TYPE ST_DivertConfig :
STRUCT
 	SwitchOpMode         						: E_SwitchOpMode;
	IntervalToDivert							: UDINT := 1;
	MaxAllowedDivertCount						: UDINT	:= 0;
	MaxAllowedCountOnShortcut					: UDINT := 2;
	CurrentFunctionCoeffA						: LREAL := 0.63;
	CurrentFunctionCoeffB						: LREAL := 0.62;
	CurrentFunctionCoeffC						: LREAL := 5;
END_STRUCT
END_TYPE;

(* stored: Version 1.1.0.1
   DUT ST_DivertConfig: Id {f50f2845-a71f-0dc3-1470-052cc68dd787} *)
